.. _Apache-2.0: https://www.apache.org/licenses/LICENSE-2.0

.. </legal notes>



*)

METHOD lengthIsBetween
VAR_INPUT
	(* current string to check *)
	stringToCheck		:POINTER TO BYTE;
	(* lower limit of the string length *)
	minLength			:UDINT;
	(* upper limit of the string length *)
	maxLength			:UDINT;
	(* string length units of measurement *)
	stringLengthUnit	:UnicodeStringLengthUnit;
	(* message if the assertion is false *)
	message				:AssertMessage;
END_VAR
VAR
	(* length of current string to check in bytes *)
	stringToCheckByteCount		:UDINT;
	(* length of current string to check in characters *)
	stringToCheckCodePointCount	:UDINT;
	
	normalizedStringBuffer :POINTER TO BYTE; 
	bufferSize :UDINT;
	normalizedLength :UDINT;
	width :DINT;
	visibleCharacters :UDINT := 0;
END_VAR
VAR CONSTANT
	(*After decomposition one codepoint can extend up to 4 codepoints*)
	NORMALIZATION_FACTOR :UDINT := 4;
END_VAR
IF minLength > maxLength THEN
	THIS^.assertionWasWrong(message, THIS^.getDebugInfo('lengthIsBetween'));
	RETURN;
END_IF

CNM_UnicodeUtilities.GetUtf8StringLength(
	stringToCheck,
	byteCount => stringToCheckByteCount,
	characterCount => stringToCheckCodePointCount
);

// check if string is empty
IF (stringToCheckByteCount = 0) THEN
	IF (minLength > 0) THEN
		THIS^.assertionWasWrong(message, THIS^.getDebugInfo('lengthIsBetween'));
	END_IF
	RETURN;
END_IF

CASE (stringLengthUnit) OF
UnicodeStringLengthUnit.BYTES:
	IF (stringToCheckByteCount < minLength OR_ELSE stringToCheckByteCount > maxLength) THEN
		THIS^.assertionWasWrong(message, THIS^.getDebugInfo('lengthIsBetween'));
	END_IF

UnicodeStringLengthUnit.CHARACTERS:
	IF (stringToCheckCodePointCount < minLength OR_ELSE stringToCheckCodePointCount > maxLength) THEN
		THIS^.assertionWasWrong(message, THIS^.getDebugInfo('lengthIsBetween'));
	END_IF	
	
UnicodeStringLengthUnit.CHARACTERS_NFC:
	// string size cant increase with NFC
	normalizedStringBuffer := __NEW(BYTE, (stringToCheckByteCount + 1));
	IF normalizedStringBuffer = 0 THEN
		THIS^.assertionWasWrong(message, THIS^.getDebugInfo('lengthIsBetween, malloc failed'));
		RETURN;
	END_IF
	
	bufferSize := stringToCheckByteCount + 1; // stringsize + NULL terminator
	
	CNM_UnicodeUtilities.NormalizeUtf8String(
		utf8StringBuffer := stringToCheck,
		normalForm := CNM_UnicodeUtilities.NormalizationForm.NFC,
		normalizedStringBuffer := normalizedStringBuffer,
		bufferSize := bufferSize,
		normalizedStringLength => normalizedLength
	);
	
	CNM_UnicodeUtilities.GetUtf8StringLength(
		stringAddress := normalizedStringBuffer,
		characterCount => stringToCheckCodePointCount
	);
	
	__DELETE(normalizedStringBuffer);
	
	IF (stringToCheckCodePointCount < minLength OR_ELSE stringToCheckCodePointCount > maxLength) THEN
		THIS^.assertionWasWrong(message, THIS^.getDebugInfo('lengthIsBetween'));
	END_IF
	
UnicodeStringLengthUnit.CHARACTERS_NFD:
	// string size can increase with NFD
	normalizedStringBuffer := __NEW(BYTE, (stringToCheckByteCount * NORMALIZATION_FACTOR + 1));
	IF normalizedStringBuffer = 0 THEN
		THIS^.assertionWasWrong(message, THIS^.getDebugInfo('lengthIsBetween, malloc failed'));
		RETURN;
	END_IF
	
	bufferSize := stringToCheckByteCount * NORMALIZATION_FACTOR + 1; // stringsize (can increase for NFD) + NULL terminator
	
	CNM_UnicodeUtilities.NormalizeUtf8String(
		utf8StringBuffer := stringToCheck,
		normalForm := CNM_UnicodeUtilities.NormalizationForm.NFD,
		normalizedStringBuffer := normalizedStringBuffer,
		bufferSize := bufferSize,
		normalizedStringLength => normalizedLength
	);
	
	CNM_UnicodeUtilities.GetUtf8StringLength(
		stringAddress := normalizedStringBuffer,
		characterCount => stringToCheckCodePointCount
	);
	
	__DELETE(normalizedStringBuffer);
	
	IF (stringToCheckCodePointCount < minLength OR_ELSE stringToCheckCodePointCount > maxLength) THEN
		THIS^.assertionWasWrong(message, THIS^.getDebugInfo('lengthIsBetween'));
	END_IF
	
UnicodeStringLengthUnit.VISIBLE_CHARACTERS:
	CNM_UnicodeUtilities.GetUtf8StringWidth(stringToCheck, visibleCharacters => visibleCharacters);
	IF (visibleCharacters < minLength) OR_ELSE (visibleCharacters > maxLength) THEN
		THIS^.assertionWasWrong(message, THIS^.getDebugInfo('lengthIsBetween'));
	END_IF 
	
UnicodeStringLengthUnit.WIDTH:
	width := CNM_UnicodeUtilities.GetUtf8StringWidth(stringToCheck);
	IF ((
			width < 0
		) OR_ELSE (
			TO_UDINT(width) < minLength
		) OR_ELSE (
			TO_UDINT(width) > maxLength)
	) THEN
		THIS^.assertionWasWrong(message, THIS^.getDebugInfo('lengthIsBetween'));
	END_IF
ELSE
	; // do nothing
END_CASE
END_METHOD

(*

## Short summary
This assertion method checks if the current string ``stringToCheck`` length is equal to ``expectedLength``.
Processed strings must be in UTF-8 encoding

**Attention:** 
	All strings are handled as null-terminated byte streams

.. <legal notes>

legal notes
=================
| SPDX-FileCopyrightText: © 2024 ekvip automation GmbH <info@ekvip.de>
| SPDX-License-Identifier: Apache-2.0
| For details check: Apache-2.0_

.. _Apache-2.0: https://www.apache.org/licenses/LICENSE-2.0

.. </legal notes>



*)

METHOD lengthIsExact
VAR_INPUT
	(* current string to check *)
	stringToCheck		:POINTER TO BYTE;
	(* expected length of ``stringToCheck`` *)
	expectedLength		:UDINT;
	(* string length units of measurement *)
	stringLengthUnit	:UnicodeStringLengthUnit;
	(* message if the assertion is false *)
	message				:AssertMessage;
END_VAR
VAR
	(* length of current string to check in bytes *)
	stringToCheckByteCount		:UDINT;
	(* length of current string to check in characters *)
	stringToCheckCodePointCount	:UDINT;
	
	normalizedStringBuffer :POINTER TO BYTE; 
	bufferSize :UDINT;
	normalizedLength :UDINT;
	width :DINT;
	visibleCharacters :UDINT := 0;
END_VAR
VAR CONSTANT
	(*After decomposition one codepoint can extend up to 4 codepoints*)
	NORMALIZATION_FACTOR :UDINT := 4;
END_VAR
CNM_UnicodeUtilities.GetUtf8StringLength(
	stringToCheck,
	byteCount => stringToCheckByteCount,
	characterCount => stringToCheckCodePointCount
);

// check if string is empty
IF (stringToCheckByteCount = 0) THEN
	IF (expectedLength <> 0) THEN
		THIS^.assertionWasWrong(message, THIS^.getDebugInfo('LengthIsExact'));
	END_IF
	RETURN;
END_IF

CASE (stringLengthUnit) OF
UnicodeStringLengthUnit.BYTES:
	IF (stringToCheckByteCount <> expectedLength) THEN
		THIS^.assertionWasWrong(message, THIS^.getDebugInfo('LengthIsExact'));
	END_IF

UnicodeStringLengthUnit.CHARACTERS:
	IF (stringToCheckCodePointCount <> expectedLength) THEN
		THIS^.assertionWasWrong(message, THIS^.getDebugInfo('LengthIsExact'));
	END_IF	
	
UnicodeStringLengthUnit.CHARACTERS_NFC:
	// string size cant increase with NFC
	normalizedStringBuffer := __NEW(BYTE, (stringToCheckByteCount+1));
	IF normalizedStringBuffer = 0 THEN
		THIS^.assertionWasWrong(message, THIS^.getDebugInfo('lengthIsExact, malloc failed'));
		RETURN;
	END_IF
	bufferSize := stringToCheckByteCount + 1; // stringsize + NULL terminator
	
	CNM_UnicodeUtilities.NormalizeUtf8String(
		utf8StringBuffer := stringToCheck,
		normalForm := CNM_UnicodeUtilities.NormalizationForm.NFC,
		normalizedStringBuffer := normalizedStringBuffer,
		bufferSize := bufferSize,
		normalizedStringLength => normalizedLength
	);
	
	CNM_UnicodeUtilities.GetUtf8StringLength(
		stringAddress := normalizedStringBuffer,
		characterCount => stringToCheckCodePointCount
	);
	
	__DELETE(normalizedStringBuffer);
	
	IF (stringToCheckCodePointCount <> expectedLength) THEN
		THIS^.assertionWasWrong(message, THIS^.getDebugInfo('LengthIsExact'));
	END_IF
	
UnicodeStringLengthUnit.CHARACTERS_NFD:
	// string size can increase with NFD
	normalizedStringBuffer := __NEW(BYTE, (stringToCheckByteCount * NORMALIZATION_FACTOR + 1));
	IF normalizedStringBuffer = 0 THEN
		THIS^.assertionWasWrong(message, THIS^.getDebugInfo('lengthIsExact, malloc failed'));
		RETURN;
	END_IF
	bufferSize := stringToCheckByteCount * NORMALIZATION_FACTOR + 1; // stringsize can increase for NFD + NULL terminator
	
	CNM_UnicodeUtilities.NormalizeUtf8String(
		utf8StringBuffer := stringToCheck,
		normalForm := CNM_UnicodeUtilities.NormalizationForm.NFD,
		normalizedStringBuffer := normalizedStringBuffer,
		bufferSize := bufferSize,
		normalizedStringLength => normalizedLength
	);
	
	CNM_UnicodeUtilities.GetUtf8StringLength(
		stringAddress := normalizedStringBuffer,
		characterCount => stringToCheckCodePointCount
	);
	
	__DELETE(normalizedStringBuffer);
	
	IF (stringToCheckCodePointCount <> expectedLength) THEN
		THIS^.assertionWasWrong(message, THIS^.getDebugInfo('LengthIsExact'));
	END_IF
	
UnicodeStringLengthUnit.VISIBLE_CHARACTERS:
	CNM_UnicodeUtilities.GetUtf8StringWidth(stringToCheck, visibleCharacters => visibleCharacters);
	IF (visibleCharacters <> expectedLength) THEN
		THIS^.assertionWasWrong(message, THIS^.getDebugInfo('lengthIsExact'));
	END_IF
	
UnicodeStringLengthUnit.WIDTH:
	width := CNM_UnicodeUtilities.GetUtf8StringWidth(stringToCheck);
	IF ((width < 0) OR_ELSE (TO_UDINT(width) <> expectedLength)) THEN
		THIS^.assertionWasWrong(message, THIS^.getDebugInfo('LengthIsExact'));
	END_IF
ELSE
	; // do nothing
END_CASE
END_METHOD

(*

## Short summary
This assertion method checks if the current string ``stringToCheck`` length is equal or less than to ``maxLength``.
Processed strings must be in UTF-8 encoding

**Attention:** 
	All strings are handled as null-terminated byte streams

.. <legal notes>

legal notes
=================
| SPDX-FileCopyrightText: © 2024 ekvip automation GmbH <info@ekvip.de>
| SPDX-License-Identifier: Apache-2.0
| For details check: Apache-2.0_

.. _Apache-2.0: https://www.apache.org/licenses/LICENSE-2.0

.. </legal notes>



*)

METHOD lengthIsMax
VAR_INPUT
	(* current string to check *)
	stringToCheck		:POINTER TO BYTE;
	(* upper limit of the length of ``stringToCheck`` *)
	maxLength			:UDINT;
	(* string length units of measurement *)
	stringLengthUnit	:UnicodeStringLengthUnit;
	(* message if the assertion is false *)
	message				:AssertMessage;
END_VAR
VAR
	(* length of current string to check in bytes *)
	stringToCheckByteCount		:UDINT;
	(* length of current string to check in characters *)
	stringToCheckCodePointCount	:UDINT;
	
	normalizedStringBuffer :POINTER TO BYTE; 
	bufferSize :UDINT;
	normalizedLength :UDINT;
	width :DINT;
	visibleCharacters :UDINT := 0;
END_VAR
VAR CONSTANT
	(*After decomposition one codepoint can extend up to 4 codepoints*)
	NORMALIZATION_FACTOR :UDINT := 4;
END_VAR
CNM_UnicodeUtilities.GetUtf8StringLength(
	stringToCheck,
	byteCount => stringToCheckByteCount,
	characterCount => stringToCheckCodePointCount
);

// check if string is empty
RETURN (stringToCheckByteCount = 0);

CASE (stringLengthUnit) OF
UnicodeStringLengthUnit.BYTES:
	IF (stringToCheckByteCount > maxLength) THEN
		THIS^.assertionWasWrong(message, THIS^.getDebugInfo('LengthIsMax'));
	END_IF

UnicodeStringLengthUnit.CHARACTERS:
	IF (stringToCheckCodePointCount > maxLength) THEN
		THIS^.assertionWasWrong(message, THIS^.getDebugInfo('LengthIsMax'));
	END_IF	
	
UnicodeStringLengthUnit.CHARACTERS_NFC:
	// string size cant increase with NFC
	normalizedStringBuffer := __NEW(BYTE, (stringToCheckByteCount + 1));
	IF normalizedStringBuffer = 0 THEN
		THIS^.assertionWasWrong(message, THIS^.getDebugInfo('lengthIsMax, malloc failed'));
		RETURN;
	END_IF
	
	// stringsize + NULL terminator
	bufferSize := stringToCheckByteCount + 1; 
	
	CNM_UnicodeUtilities.NormalizeUtf8String(
		utf8StringBuffer := stringToCheck,
		normalForm := CNM_UnicodeUtilities.NormalizationForm.NFC,
		normalizedStringBuffer := normalizedStringBuffer,
		bufferSize := bufferSize,
		normalizedStringLength => normalizedLength
	);
	
	CNM_UnicodeUtilities.GetUtf8StringLength(
		stringAddress := normalizedStringBuffer,
		characterCount => stringToCheckCodePointCount
	);
	
	__DELETE(normalizedStringBuffer);
	
	IF (stringToCheckCodePointCount > maxLength) THEN
		THIS^.assertionWasWrong(message, THIS^.getDebugInfo('LengthIsMax'));
	END_IF
	
UnicodeStringLengthUnit.CHARACTERS_NFD:
	// string size can increase with NFD
	normalizedStringBuffer := __NEW(BYTE, (stringToCheckByteCount * NORMALIZATION_FACTOR + 1));
	IF normalizedStringBuffer = 0 THEN
		THIS^.assertionWasWrong(message, THIS^.getDebugInfo('lengthIsMax, malloc failed'));
		RETURN;
	END_IF
	bufferSize := stringToCheckByteCount * NORMALIZATION_FACTOR + 1; // stringsize can increase for NFD + NULL terminator
	
	CNM_UnicodeUtilities.NormalizeUtf8String(
		utf8StringBuffer := stringToCheck,
		normalForm := CNM_UnicodeUtilities.NormalizationForm.NFD,
		normalizedStringBuffer := normalizedStringBuffer,
		bufferSize := bufferSize,
		normalizedStringLength => normalizedLength
	);
	
	CNM_UnicodeUtilities.GetUtf8StringLength(
		stringAddress := normalizedStringBuffer,
		characterCount => stringToCheckCodePointCount
	);
	
	__DELETE(normalizedStringBuffer);
	
	IF (stringToCheckCodePointCount > maxLength) THEN
		THIS^.assertionWasWrong(message, THIS^.getDebugInfo('LengthIsMax'));
	END_IF
	
UnicodeStringLengthUnit.VISIBLE_CHARACTERS:
	CNM_UnicodeUtilities.GetUtf8StringWidth(stringToCheck, visibleCharacters => visibleCharacters);
	IF (visibleCharacters > maxLength) THEN
		THIS^.assertionWasWrong(message, THIS^.getDebugInfo('lengthIsMax'));
	END_IF
	
UnicodeStringLengthUnit.WIDTH:
	width := CNM_UnicodeUtilities.GetUtf8StringWidth(stringToCheck);
	IF ((width < 0) OR_ELSE (TO_UDINT(width) > maxLength)) THEN
		THIS^.assertionWasWrong(message, THIS^.getDebugInfo('LengthIsMax'));
	END_IF
ELSE
	; // do nothing
END_CASE
END_METHOD

(*

## Short summary
This assertion method checks if the current string ``stringToCheck`` length is equal or grater than to ``minLength``.
Processed strings must be in UTF-8 encoding

**Attention:** 
	All strings are handled as null-terminated byte streams

.. <legal notes>

legal notes
=================
| SPDX-FileCopyrightText: © 2024 ekvip automation GmbH <info@ekvip.de>
| SPDX-License-Identifier: Apache-2.0
| For details check: Apache-2.0_

.. _Apache-2.0: https://www.apache.org/licenses/LICENSE-2.0

.. </legal notes>



*)

METHOD lengthIsMin
VAR_INPUT
	(* current string to check *)
	stringToCheck		:POINTER TO BYTE;
	(* lower limit of the length of ``stringToCheck`` *)
	minLength			:UDINT;
	(* string length units of measurement *)
	stringLengthUnit	:UnicodeStringLengthUnit;
	(* message if the assertion is false *)
	message				:AssertMessage;
END_VAR
VAR
	(* length of current string to check in bytes *)
	stringToCheckByteCount		:UDINT;
	(* length of current string to check in characters *)
	stringToCheckCodePointCount	:UDINT;
	normalizedStringBuffer :POINTER TO BYTE; 
	bufferSize :UDINT;
	normalizedLength :UDINT;
	width :DINT;
	visibleCharacters :UDINT := 0;
END_VAR
VAR CONSTANT
	(*After decomposition one codepoint can extend up to 4 codepoints*)
	NORMALIZATION_FACTOR :UDINT := 4;
END_VAR
CNM_UnicodeUtilities.GetUtf8StringLength(
	stringToCheck,
	byteCount => stringToCheckByteCount,
	characterCount => stringToCheckCodePointCount
);

// check if string is empty
IF (stringToCheckByteCount = 0) THEN
	IF (minLength > 0) THEN
		THIS^.assertionWasWrong(message, THIS^.getDebugInfo('LengthIsMin'));
	END_IF
	RETURN;
END_IF

CASE (stringLengthUnit) OF
UnicodeStringLengthUnit.BYTES:
	IF (stringToCheckByteCount < minLength) THEN
		THIS^.assertionWasWrong(message, THIS^.getDebugInfo('LengthIsMin'));
	END_IF

UnicodeStringLengthUnit.CHARACTERS:
	IF (stringToCheckCodePointCount < minLength) THEN
		THIS^.assertionWasWrong(message, THIS^.getDebugInfo('LengthIsMin'));
	END_IF	
	
UnicodeStringLengthUnit.CHARACTERS_NFC:
	// string size cant increase with NFC
	normalizedStringBuffer := __NEW(BYTE, (stringToCheckByteCount + 1));
	IF normalizedStringBuffer = 0 THEN
		THIS^.assertionWasWrong(message, THIS^.getDebugInfo('lengthIsMin, malloc failed'));
		RETURN;
	END_IF
	bufferSize := stringToCheckByteCount + 1; // stringsize + NULL terminator
	
	CNM_UnicodeUtilities.NormalizeUtf8String(
		utf8StringBuffer := stringToCheck,
		normalForm := CNM_UnicodeUtilities.NormalizationForm.NFC,
		normalizedStringBuffer := normalizedStringBuffer,
		bufferSize := bufferSize,
		normalizedStringLength => normalizedLength
	);
	
	CNM_UnicodeUtilities.GetUtf8StringLength(
		stringAddress := normalizedStringBuffer,
		characterCount => stringToCheckCodePointCount
	);
	
	__DELETE(normalizedStringBuffer);
	
	IF (stringToCheckCodePointCount < minLength) THEN
		THIS^.assertionWasWrong(message, THIS^.getDebugInfo('LengthIsMin'));
	END_IF
	
UnicodeStringLengthUnit.CHARACTERS_NFD:
	// string size can increase with NFD
	normalizedStringBuffer := __NEW(BYTE, (stringToCheckByteCount * NORMALIZATION_FACTOR + 1));
	IF normalizedStringBuffer = 0 THEN
		THIS^.assertionWasWrong(message, THIS^.getDebugInfo('lengthIsMin, malloc failed'));
		RETURN;
	END_IF
	bufferSize := stringToCheckByteCount * NORMALIZATION_FACTOR + 1; // stringsize can increase for NFD + NULL terminator
	
	CNM_UnicodeUtilities.NormalizeUtf8String(
		utf8StringBuffer := stringToCheck,
		normalForm := CNM_UnicodeUtilities.NormalizationForm.NFD,
		normalizedStringBuffer := normalizedStringBuffer,
		bufferSize := bufferSize,
		normalizedStringLength => normalizedLength
	);
	
	CNM_UnicodeUtilities.GetUtf8StringLength(
		stringAddress := normalizedStringBuffer,
		characterCount => stringToCheckCodePointCount
	);
	
	__DELETE(normalizedStringBuffer);
	
	IF (stringToCheckCodePointCount < minLength) THEN
		THIS^.assertionWasWrong(message, THIS^.getDebugInfo('LengthIsMin'));
	END_IF
	
UnicodeStringLengthUnit.VISIBLE_CHARACTERS:
	CNM_UnicodeUtilities.GetUtf8StringWidth(stringToCheck, visibleCharacters => visibleCharacters);
	IF (visibleCharacters < minLength)THEN
		THIS^.assertionWasWrong(message, THIS^.getDebugInfo('lengthIsMin'));
	END_IF
	
UnicodeStringLengthUnit.WIDTH:
	width := CNM_UnicodeUtilities.GetUtf8StringWidth(stringToCheck);
	IF ((width < 0) OR_ELSE (TO_UDINT(width) < minLength)) THEN
		THIS^.assertionWasWrong(message, THIS^.getDebugInfo('LengthIsMin'));
	END_IF
ELSE
	; // do nothing
END_CASE
END_METHOD

(*

## Short summary
This assertion method checks if the current string ``stringToCheck`` starts with string ``start``.
Processed strings must be in UTF-8 encoding

**Attention:** 
	All strings are handled as null-terminated byte streams

.. <legal notes>

legal notes
=================
| SPDX-FileCopyrightText: © 2024 ekvip automation GmbH <info@ekvip.de>
| SPDX-License-Identifier: Apache-2.0
| For details check: Apache-2.0_

.. _Apache-2.0: https://www.apache.org/licenses/LICENSE-2.0

.. </legal notes>



*)

METHOD startsWith
VAR_INPUT
	(* current string to check *)
	stringToCheck	:POINTER TO BYTE;
	(* expected start of ``stringToCheck`` *)
	start			:POINTER TO BYTE;
	(* ``TRUE`` means ignore cases; ``FALSE`` means that cases must be equal too *)
	ignoreCases		:BOOL;
	(* ``TRUE`` means truncation of spaces on the left side of ``stringToCheck``*)
	trim		:BOOL;
	(* message if the assertion is false *)
	message			:AssertMessage;
	(*normalize both strings for check*)
	normalizeStrings :BOOL := TRUE;
END_VAR
VAR
	(* length of ``stringToCheck`` in bytes *)
	lengthStringToCheckInByte	:UDINT;	
	(* length of ``searchString`` in bytes *)
	lengthSearchStringInByte	:UDINT;
	(* DWORD array we use to check *)
	usedCodePointsToCheck, normalizedUsedCodePointsToCheck :POINTER TO CNM_UnicodeUtilities.UnicodeCodePoint;
	usedCodePointToCheckCount	:UDINT;
	
	(* DWORD array we use to compare *)
	usedStartCodePoints, normalizedUsedStartCodePoints :POINTER TO CNM_UnicodeUtilities.UnicodeCodePoint;
	usedStartCodePointCount		:UDINT;
END_VAR
VAR CONSTANT
	(*After decomposition one codepoint can extend up to 4 codepoints*)
	NORMALIZATION_FACTOR :UDINT := 4;
END_VAR
CNM_UnicodeUtilities.GetUtf8StringLength(stringAddress := stringToCheck, byteCount => lengthStringToCheckInByte);
CNM_UnicodeUtilities.GetUtf8StringLength(stringAddress := start, byteCount => lengthSearchStringInByte);

IF (((
		NOT normalizeStrings 
	) OR ( 
		lengthStringToCheckInByte = 0
	) OR (
		lengthSearchStringInByte = 0
	)) AND_THEN(
		NOT THIS^.isContainsCheckNecessary(
			stringToCheck		:= stringToCheck,
			searchString		:= start,
			lengthStringToCheck	:= lengthStringToCheckInByte,
			lengthSearchString	:= lengthSearchStringInByte,
			additionalText		:= THIS^.getDebugInfo('startsWith'),
			message				:= message
		) 
	)
) THEN
	RETURN;
END_IF

usedCodePointsToCheck := __NEW(CNM_UnicodeUtilities.UnicodeCodePoint, lengthStringToCheckInByte);
IF (usedCodePointsToCheck = 0) THEN
	THIS^.assertionWasWrong(message, THIS^.getDebugInfo('startsWith, malloc failed'));
	RETURN;
END_IF

usedStartCodePoints := __NEW(CNM_UnicodeUtilities.UnicodeCodePoint, lengthSearchStringInByte);
IF (usedStartCodePoints = 0) THEN
	__DELETE(usedCodePointsToCheck);
	THIS^.assertionWasWrong(message, THIS^.getDebugInfo('startsWith, malloc failed'));
	RETURN;
END_IF

(* convert ``stringToCheck`` to code points *)
CNM_UnicodeUtilities.GetCodepointsFromUtf8String(
	utf8StringAddress := stringToCheck, 
	utf8StringByteCount := lengthStringToCheckInByte, 
	codePointBuffer := usedCodePointsToCheck,
	bufferSize := SIZEOF(CNM_UnicodeUtilities.UnicodeCodePoint)*lengthStringToCheckInByte, 
	codePointsCount => usedCodePointToCheckCount);

(* convert ``searchString`` to code points *)
CNM_UnicodeUtilities.GetCodepointsFromUtf8String(
	utf8StringAddress 	:= start, 
	utf8StringByteCount := lengthSearchStringInByte, 
	codePointBuffer	:= usedStartCodePoints,
	bufferSize := SIZEOF(CNM_UnicodeUtilities.UnicodeCodePoint)*lengthSearchStringInByte,
	codePointsCount => usedStartCodePointCount);



IF normalizeStrings THEN
	normalizedUsedCodePointsToCheck := __NEW(
		CNM_UnicodeUtilities.UnicodeCodePoint,
		(lengthStringToCheckInByte * NORMALIZATION_FACTOR)
	);
	IF (normalizedUsedCodePointsToCheck = 0) THEN
		THIS^.assertionWasWrong(message, THIS^.getDebugInfo('startsWith, malloc failed'));
		__DELETE(usedCodePointsToCheck);
		__DELETE(usedStartCodePoints);
		RETURN;
	END_IF
	normalizedUsedStartCodePoints := __NEW(
		CNM_UnicodeUtilities.UnicodeCodePoint,
		(lengthSearchStringInByte * NORMALIZATION_FACTOR)
	);
	IF (normalizedUsedStartCodePoints = 0) THEN
		THIS^.assertionWasWrong(message, THIS^.getDebugInfo('startsWith, malloc failed'));
		__DELETE(usedCodePointsToCheck);
		__DELETE(usedStartCodePoints);
		__DELETE(normalizedUsedCodePointsToCheck);	
		RETURN;
	END_IF

	CNM_UnicodeUtilities.NormalizeCodepointsFormD(
		codePoints := usedCodePointsToCheck,
		codePointsCount := usedCodePointToCheckCount,
		normalizedCodepoints := normalizedUsedCodePointsToCheck,
		bufferSize := (lengthStringToCheckInByte * NORMALIZATION_FACTOR) * SIZEOF(CNM_UnicodeUtilities.UnicodeCodePoint),
		normalizedCodepointsCount => usedCodePointToCheckCount
	);
	__DELETE(usedCodePointsToCheck);
	usedCodePointsToCheck := normalizedUsedCodePointsToCheck;
	
	CNM_UnicodeUtilities.NormalizeCodepointsFormD(
		codePoints := usedStartCodePoints,
		codePointsCount := usedStartCodePointCount,
		normalizedCodepoints := normalizedUsedStartCodePoints,
		bufferSize := (lengthSearchStringInByte * NORMALIZATION_FACTOR) * SIZEOF(CNM_UnicodeUtilities.UnicodeCodePoint),
		normalizedCodepointsCount => usedStartCodePointCount
	);
	__DELETE(usedStartCodePoints);
	usedStartCodePoints := normalizedUsedStartCodePoints;
END_IF

IF (trim) THEN
	CNM_UnicodeUtilities.TrimLeftCodepoints(
		codepoints := usedStartCodePoints,
		codepointCount := usedStartCodePointCount,
		newCodepointCount => usedStartCodePointCount
	);
	CNM_UnicodeUtilities.TrimLeftCodepoints(
		codepoints := usedCodePointsToCheck,
		codepointCount := usedCodePointToCheckCount,
		newCodepointCount => usedCodePointToCheckCount
	);
END_IF

IF (ignoreCases) THEN
	CNM_UnicodeUtilities.GetUpperCaseForCodepoint(usedCodePointsToCheck, usedCodePointToCheckCount);
	CNM_UnicodeUtilities.GetUpperCaseForCodepoint(usedStartCodePoints, usedStartCodePointCount);
END_IF

IF (Tc2_System.MEMCMP(
		usedCodePointsToCheck,
		usedStartCodePoints, 
		usedStartCodePointCount*SIZEOF(CNM_UnicodeUtilities.UnicodeCodePoint)
	) <> CNM_ReturnTypes.ComparationResult.EQUAL
) THEN
	THIS^.assertionWasWrong(message, THIS^.getDebugInfo('startsWith'));
END_IF;

__DELETE(usedCodePointsToCheck);
__DELETE(usedStartCodePoints);
END_METHOD

END_FUNCTION_BLOCK

// ---- Assertor/Assertions/StringAssertion/Unicode/Classes/UnicodeAssertions.TcPOU
(*

## Short summary
Class provides assert statements
for UTF-8 and UTF-16 strings with an undefined length.

**Attention:** 
	All strings are handled as null terminated byte/word streams.
	For UTF-8 is end of the string 16#00
	For UTF-16 is end of the string 16#00_00

**Attention:** 
	The interface `IUnicodeAssertions` uses ``ANY_STRING``, 
	for this it's not possible to use literals/constants,
	because for ``ANY`` types generates the compiler ``__SYSTEM.AnyType``
	and ``__SYSTEM.AnyType`` contains a pointer  

.. <legal notes>

legal notes
=================
| SPDX-FileCopyrightText: © 2022 ekvip automation GmbH <info@ekvip.de>
| SPDX-License-Identifier: Apache-2.0
| For details check: Apache-2.0_

.. _Apache-2.0: https://www.apache.org/licenses/LICENSE-2.0

.. </legal notes>



*)

{attribute 'reflection'}
FUNCTION_BLOCK INTERNAL UnicodeAssertions EXTENDS AbstractAssertion IMPLEMENTS IUnicodeStringAssertions
VAR
	(* class to handle the utf 8 string assertions *)  
	utf8Assertions	:Utf8StringPointerAssertions();
	(* class to handle the utf 16 string assertions *)  
	utf16Assertions		:Utf16StringPointerAssertions();	
END_VAR

(*

## Short summary
This abstract property returns the class name of the concrete object, 
It's for debugging purpose

.. <legal notes>

legal notes
=================
| SPDX-FileCopyrightText: © 2022 ekvip automation GmbH <info@ekvip.de>
| SPDX-License-Identifier: Apache-2.0
| For details check: Apache-2.0_

.. _Apache-2.0: https://www.apache.org/licenses/LICENSE-2.0

.. </legal notes>

*)

PROPERTY className :CNM_AbstractObject.ClassName
GET
className := 'CNM_Assertor.UnicodeAssertions';
END_GET
END_PROPERTY

(*

## Short summary
This assertion method checks if the current string ``stringToCheck`` contains the search string

**Attention:** 
	All strings are handled as null terminated byte/word streams.
	For UTF-8 is end of the string 16#00
	For UTF-16 is end of the string 16#00_00

**Attention:** 
	The interface `IUnicodeAssertions` uses ``ANY_STRING``, 
	for this it's not possible to use literals/constants,
	because for ``ANY`` types generates the compiler ``__SYSTEM.AnyType``
	and ``__SYSTEM.AnyType`` contains a pointer  

.. <legal notes>

legal notes
=================
| SPDX-FileCopyrightText: © 2022 ekvip automation GmbH <info@ekvip.de>
| SPDX-License-Identifier: Apache-2.0
| For details check: Apache-2.0_

.. _Apache-2.0: https://www.apache.org/licenses/LICENSE-2.0

.. </legal notes>



*)

METHOD contains
VAR_INPUT
	(* current string to check *)
	stringToCheck	:ANY_STRING;
	(* string must be found in ``stringToCheck`` *)
	searchString	:ANY_STRING;
	(* message if the assertion is false *)
	message			:AssertMessage;
	(* ``TRUE`` means ignore cases; ``FALSE`` means cases must be equal too *)
	ignoreCases		:BOOL := FALSE;
	(*normalize both strings for check*)
	normalizeStrings :BOOL := TRUE;
END_VAR
IF ((
		stringToCheck.TypeClass <> searchString.TypeClass
	) OR_ELSE (
		stringToCheck.diSize = 0 
	) OR_ELSE ( 
		searchString.diSize = 0 
	)
) THEN
	THIS^.assertionWasWrong(message, THIS^.getDebugInfo('contains'));
	RETURN;
END_IF

CASE stringToCheck.TypeClass OF
TYPE_CLASS.TYPE_STRING:
	THIS^.utf8Assertions.contains(
		stringToCheck := stringToCheck.pValue,
		searchString := searchString.pValue,
		ignoreCases := ignoreCases,
		message := message
	);
TYPE_CLASS.TYPE_WSTRING:
	THIS^.utf16Assertions.contains(
		stringToCheck := stringToCheck.pValue,
		searchString := searchString.pValue,
		ignoreCases := ignoreCases,
		message := message,
		normalizeStrings := normalizeStrings
	);
ELSE
	; // do nothing
END_CASE
END_METHOD

(*

## Short summary
This assertion method checks if the current string ``stringToCheck`` not contains the search string

**Attention:** 
	All strings are handled as null terminated byte/word streams.
	For UTF-8 is end of the string 16#00
	For UTF-16 is end of the string 16#00_00

**Attention:** 
	The interface `IUnicodeAssertions` uses ``ANY_STRING``, 
	for this it's not possible to use literals/constants,
	because for ``ANY`` types generates the compiler ``__SYSTEM.AnyType``
	and ``__SYSTEM.AnyType`` contains a pointer  

.. <legal notes>

legal notes
=================
| SPDX-FileCopyrightText: © 2022 ekvip automation GmbH <info@ekvip.de>
| SPDX-License-Identifier: Apache-2.0
| For details check: Apache-2.0_

.. _Apache-2.0: https://www.apache.org/licenses/LICENSE-2.0

.. </legal notes>



*)

METHOD containsNo
VAR_INPUT
	(* current string to check *)
	stringToCheck	:ANY_STRING;
	(* string that must not be found in ``stringToCheck`` *)
	searchString	:ANY_STRING;
	(* message if the assertion is false *)
	message			:AssertMessage;
	(* ``TRUE`` means ignore cases; ``FALSE`` means cases must be equal too *)
	ignoreCases		:BOOL := FALSE;
	(*normalize both strings for check*)
	normalizeStrings :BOOL := TRUE;
END_VAR
IF ((
		stringToCheck.TypeClass <> searchString.TypeClass
	) OR_ELSE ( 
		stringToCheck.diSize = 0 
	) OR_ELSE ( 
		searchString.diSize = 0 
	)
) THEN
	THIS^.assertionWasWrong(message, THIS^.getDebugInfo('containsNo'));
	RETURN;
END_IF

CASE stringToCheck.TypeClass OF
TYPE_CLASS.TYPE_STRING:
	THIS^.utf8Assertions.containsNo(
		stringToCheck := stringToCheck.pValue,
		searchString := searchString.pValue,
		ignoreCases := ignoreCases,
		message := message
	);
TYPE_CLASS.TYPE_WSTRING:
	THIS^.utf16Assertions.containsNo(
		stringToCheck := stringToCheck.pValue,
		searchString := searchString.pValue,
		ignoreCases := ignoreCases,
		message := message,
		normalizeStrings := normalizeStrings
	);
ELSE
	; // do nothing
END_CASE
END_METHOD

(*

## Short summary
This assertion method checks if the current string ``stringToCheck`` ends with ``end``

**Attention:** 
	All strings are handled as null terminated byte/word streams.
	For UTF-8 is end of the string 16#00
	For UTF-16 is end of the string 16#00_00

**Attention:** 
	The interface `IUnicodeAssertions` uses ``ANY_STRING``, 
	for this it's not possible to use literals/constants,
	because for ``ANY`` types generates the compiler ``__SYSTEM.AnyType``
	and ``__SYSTEM.AnyType`` contains a pointer  

**Attention:** 
	end of the string is **ALWAYS** the right side of the string 
	even for writings which written from right to left like Hebrew or Arabic

.. <legal notes>

legal notes
=================
| SPDX-FileCopyrightText: © 2022 ekvip automation GmbH <info@ekvip.de>
| SPDX-License-Identifier: Apache-2.0
| For details check: Apache-2.0_

.. _Apache-2.0: https://www.apache.org/licenses/LICENSE-2.0

.. </legal notes>



*)

METHOD endsWith
VAR_INPUT
	(* current string to check *)
	stringToCheck	:ANY_STRING;
	(* expected end of ``stringToCheck`` *)
	end				:ANY_STRING;
	(* message if the assertion is false *)
	message			:AssertMessage;
	(* ``TRUE`` means ignore cases; ``FALSE`` means cases must be equal too *)
	ignoreCases		:BOOL := FALSE;
	(* ``TRUE`` means truncation of spaces on the right side of ``stringToCheck``*)
	trim			:BOOL := FALSE;
	(*normalize both strings for check*)
	normalizeStrings :BOOL := TRUE;
END_VAR
IF ((
		stringToCheck.TypeClass <> end.TypeClass
	) OR_ELSE (
		 stringToCheck.diSize = 0
	) OR_ELSE (
		 end.diSize = 0
	)
) THEN
	THIS^.assertionWasWrong(message, THIS^.getDebugInfo('endsWith'));
	RETURN;
END_IF

CASE stringToCheck.TypeClass OF
TYPE_CLASS.TYPE_STRING:
	THIS^.utf8Assertions.endsWith(
		stringToCheck := stringToCheck.pValue,
		end := end.pValue,
		ignoreCases := ignoreCases,
		trim := trim,
		message := message,
		normalizeStrings := normalizeStrings
	);
TYPE_CLASS.TYPE_WSTRING:
	THIS^.utf16Assertions.endsWith(
		stringToCheck := stringToCheck.pValue,
		end := end.pValue,
		ignoreCases := ignoreCases,
		trim := trim,
		message := message,
		normalizeStrings := normalizeStrings
	);
ELSE
	; // do nothing
END_CASE
END_METHOD

(*

## Short summary
This assertion method checks if the current string ``stringToCheck`` is empty

**Attention:** 
	All strings are handled as null terminated byte/word streams.
	For UTF-8 is end of the string 16#00
	For UTF-16 is end of the string 16#00_00

**Attention:** 
	The interface `IUnicodeAssertions` uses ``ANY_STRING``, 
	for this it's not possible to use literals/constants,
	because for ``ANY`` types generates the compiler ``__SYSTEM.AnyType``
	and ``__SYSTEM.AnyType`` contains a pointer  

.. <legal notes>

legal notes
=================
| SPDX-FileCopyrightText: © 2022 ekvip automation GmbH <info@ekvip.de>
| SPDX-License-Identifier: Apache-2.0
| For details check: Apache-2.0_

.. _Apache-2.0: https://www.apache.org/licenses/LICENSE-2.0

.. </legal notes>



*)

METHOD isEmpty
VAR_INPUT
	(* current string to check *)
	stringToCheck	:ANY_STRING;
	(* message if the assertion is false *)
	message			:AssertMessage;
END_VAR
VAR CONSTANT
	(* strings are null terminated *)
	END_OF_UTF8_STRING	:BYTE := 16#00;
	(* strings are null terminated *)
	END_OF_UTF16_STRING	:WORD := 16#0000;
END_VAR
CASE stringToCheck.TypeClass OF
TYPE_CLASS.TYPE_STRING:
	IF (stringToCheck.pValue^ <> END_OF_UTF8_STRING) THEN
		THIS^.assertionWasWrong(message, THIS^.getDebugInfo('isEmpty'));
	END_IF
TYPE_CLASS.TYPE_WSTRING:
	IF (stringToCheck.pValue^ <> END_OF_UTF16_STRING) THEN
		THIS^.assertionWasWrong(message, THIS^.getDebugInfo('isEmpty'));
	END_IF
ELSE
	; // do nothing
END_CASE
END_METHOD

(*

## Short summary
This assertion method checks if the current string ``stringToCheck`` is equal to ``expected``

**Attention:** 
	All strings are handled as null terminated byte/word streams.
	For UTF-8 is end of the string 16#00
	For UTF-16 is end of the string 16#00_00

**Attention:** 
	The interface `IUnicodeAssertions` uses ``ANY_STRING``, 
	for this it's not possible to use literals/constants,
	because for ``ANY`` types generates the compiler ``__SYSTEM.AnyType``
	and ``__SYSTEM.AnyType`` contains a pointer  

.. <legal notes>

legal notes
=================
| SPDX-FileCopyrightText: © 2022 ekvip automation GmbH <info@ekvip.de>
| SPDX-License-Identifier: Apache-2.0
| For details check: Apache-2.0_

.. _Apache-2.0: https://www.apache.org/licenses/LICENSE-2.0

.. </legal notes>



*)

METHOD isEqualTo
VAR_INPUT
	(* current string to check *)
	stringToCheck	:ANY_STRING;
	(* ``stringToCheck`` must be equal to expected *)
	expected		:ANY_STRING;
	(* message if the assertion is false *)
	message			:AssertMessage;
	(* ``TRUE`` means ignore cases; ``FALSE`` means cases must be equal too *)
	ignoreCases		:BOOL := FALSE;
	(*normalize both strings for check*)
	normalizeStrings :BOOL := TRUE;
END_VAR
IF ((
		stringToCheck.TypeClass <> expected.TypeClass
	) OR_ELSE ( 
		stringToCheck.diSize = 0
	) OR_ELSE ( 
		expected.diSize = 0 
	)
) THEN
	THIS^.assertionWasWrong(message, THIS^.getDebugInfo('isEqualTo'));
	RETURN;
END_IF

CASE stringToCheck.TypeClass OF
TYPE_CLASS.TYPE_STRING:
	THIS^.utf8Assertions.isEqualTo(
		stringToCheck := stringToCheck.pValue,
		expected := expected.pValue,
		ignoreCases := ignoreCases,
		message := message
	);
TYPE_CLASS.TYPE_WSTRING:
	THIS^.utf16Assertions.isEqualTo(
		stringToCheck := stringToCheck.pValue,
		expected := expected.pValue,
		ignoreCases := ignoreCases,
		message := message,
		normalizeStrings := normalizeStrings
	);	
ELSE
	; // do nothing
END_CASE
END_METHOD

(*

## Short summary
This assertion method checks if the current string ``stringToCheck`` is not empty

**Attention:** 
	All strings are handled as null terminated byte/word streams.
	For UTF-8 is end of the string 16#00
	For UTF-16 is end of the string 16#00_00

**Attention:** 
	The interface `IUnicodeAssertions` uses ``ANY_STRING``, 
	for this it's not possible to use literals/constants,
	because for ``ANY`` types generates the compiler ``__SYSTEM.AnyType``
	and ``__SYSTEM.AnyType`` contains a pointer  

.. <legal notes>

legal notes
=================
| SPDX-FileCopyrightText: © 2022 ekvip automation GmbH <info@ekvip.de>
| SPDX-License-Identifier: Apache-2.0
| For details check: Apache-2.0_

.. _Apache-2.0: https://www.apache.org/licenses/LICENSE-2.0

.. </legal notes>



*)

METHOD isNotEmpty
VAR_INPUT
	(* current string to check *)
	stringToCheck	:ANY_STRING;
	(* message if the assertion is false *)
	message			:AssertMessage;
END_VAR
VAR CONSTANT
	(* strings are null terminated *)
	END_OF_UTF8_STRING	:BYTE := 16#00;
	(* strings are null terminated *)
	END_OF_UTF16_STRING	:WORD := 16#0000;
END_VAR
CASE stringToCheck.TypeClass OF
TYPE_CLASS.TYPE_STRING:
	IF (stringToCheck.pValue^ = END_OF_UTF8_STRING) THEN
		THIS^.assertionWasWrong(message, THIS^.getDebugInfo('isNotEmpty'));
	END_IF
TYPE_CLASS.TYPE_WSTRING:
	IF (stringToCheck.pValue^ = END_OF_UTF16_STRING) THEN
		THIS^.assertionWasWrong(message, THIS^.getDebugInfo('isNotEmpty'));
	END_IF
ELSE
	; // do nothing
END_CASE
END_METHOD

(*

## Short summary
This assertion method checks if the current string ``stringToCheck`` is not equal to ``unexpected``

**Attention:** 
	All strings are handled as null terminated byte/word streams.
	For UTF-8 is end of the string 16#00
	For UTF-16 is end of the string 16#00_00

**Attention:** 
	The interface `IUnicodeAssertions` uses ``ANY_STRING``, 
	for this it's not possible to use literals/constants,
	because for ``ANY`` types generates the compiler ``__SYSTEM.AnyType``
	and ``__SYSTEM.AnyType`` contains a pointer  

.. <legal notes>

legal notes
=================
| SPDX-FileCopyrightText: © 2022 ekvip automation GmbH <info@ekvip.de>
| SPDX-License-Identifier: Apache-2.0
| For details check: Apache-2.0_

.. _Apache-2.0: https://www.apache.org/licenses/LICENSE-2.0

.. </legal notes>



*)

METHOD isNotEqualTo
VAR_INPUT
	(* current string to check *)
	stringToCheck	:ANY_STRING;
	(* ``stringToCheck`` must be not equal to expected *)
	unexpected		:ANY_STRING;
	(* message if the assertion is false *)
	message			:AssertMessage;
	(* ``TRUE`` means ignore cases; ``FALSE`` means cases must be equal too *)
	ignoreCases		:BOOL := FALSE;
	(*normalize both strings for check*)
	normalizeStrings :BOOL := TRUE;
END_VAR
IF ((
		stringToCheck.TypeClass <> unexpected.TypeClass
	) OR_ELSE ( 
		stringToCheck.diSize = 0 
	) OR_ELSE ( 
		unexpected.diSize = 0 
	)
) THEN
	THIS^.assertionWasWrong(message, THIS^.getDebugInfo('isNotEqualTo'));
	RETURN;
END_IF

CASE stringToCheck.TypeClass OF
TYPE_CLASS.TYPE_STRING:
	THIS^.utf8Assertions.isNotEqualTo(
		stringToCheck := stringToCheck.pValue,
		unexpected := unexpected.pValue,
		ignoreCases := ignoreCases,
		message := message
	);
TYPE_CLASS.TYPE_WSTRING:
	THIS^.utf16Assertions.isNotEqualTo(
		stringToCheck := stringToCheck.pValue,
		unexpected := unexpected.pValue,
		ignoreCases := ignoreCases,
		message := message,
		normalizeStrings := normalizeStrings
	);	
ELSE
	; // do nothing
END_CASE
END_METHOD

(*

## Short summary
This assertion method checks if the current string ``stringToCheck`` is length
is between ``minLength`` and ``maxLength``

**Attention:** 
	All strings are handled as null terminated byte/word streams.
	For UTF-8 is end of the string 16#00
	For UTF-16 is end of the string 16#00_00

**Attention:** 
	The interface `IUnicodeAssertions` uses ``ANY_STRING``, 
	for this it's not possible to use literals/constants,
	because for ``ANY`` types generates the compiler ``__SYSTEM.AnyType``
	and ``__SYSTEM.AnyType`` contains a pointer  

.. <legal notes>

legal notes
=================
| SPDX-FileCopyrightText: © 2022 ekvip automation GmbH <info@ekvip.de>
| SPDX-License-Identifier: Apache-2.0
| For details check: Apache-2.0_

.. _Apache-2.0: https://www.apache.org/licenses/LICENSE-2.0

.. </legal notes>



*)

METHOD lengthIsBetween
VAR_INPUT
	(* current string to check *)
	stringToCheck	:ANY_STRING;
	(* lower limit of the string length *)
	minLength		:UDINT;
	(* upper limit of the string length *)
	maxLength		:UDINT;
	(* string length units of measurement *)
	stringLengthUnit	:UnicodeStringLengthUnit;
	(* message if the assertion is false *)
	message			:AssertMessage;
END_VAR
CASE stringToCheck.TypeClass OF
TYPE_CLASS.TYPE_STRING:
	THIS^.utf8Assertions.lengthIsBetween(
		stringToCheck	:= stringToCheck.pValue,
		minLength		:= minLength,
		maxLength		:= maxLength,
		stringLengthUnit := stringLengthUnit,
		message			:= message		
	);
TYPE_CLASS.TYPE_WSTRING:
	THIS^.utf16Assertions.lengthIsBetween(
		stringToCheck	:= stringToCheck.pValue,
		minLength		:= minLength,
		maxLength		:= maxLength,
		stringLengthUnit := stringLengthUnit,
		message			:= message
	);
ELSE
	; // do nothing
END_CASE
END_METHOD

(*

## Short summary
This assertion method checks if the current string ``stringToCheck`` is length
is equal to ``expectedLength``

**Attention:** 
	All strings are handled as null terminated byte/word streams.
	For UTF-8 is end of the string 16#00
	For UTF-16 is end of the string 16#00_00

**Attention:** 
	The interface `IUnicodeAssertions` uses ``ANY_STRING``, 
	for this it's not possible to use literals/constants,
	because for ``ANY`` types generates the compiler ``__SYSTEM.AnyType``
	and ``__SYSTEM.AnyType`` contains a pointer  

.. <legal notes>

legal notes
=================
| SPDX-FileCopyrightText: © 2022 ekvip automation GmbH <info@ekvip.de>
| SPDX-License-Identifier: Apache-2.0
| For details check: Apache-2.0_

.. _Apache-2.0: https://www.apache.org/licenses/LICENSE-2.0

.. </legal notes>



*)

METHOD lengthIsExact
VAR_INPUT
	(* current string to check *)
	stringToCheck	:ANY_STRING;
	(* expected length of ``stringToCheck`` *)
	expectedLength	:UDINT;
	(* string length units of measurement *)
	stringLengthUnit	:UnicodeStringLengthUnit;
	(* message if the assertion is false *)
	message			:AssertMessage;
END_VAR
CASE stringToCheck.TypeClass OF
TYPE_CLASS.TYPE_STRING:
	THIS^.utf8Assertions.lengthIsExact(
		stringToCheck	:= stringToCheck.pValue,
		expectedLength	:= expectedLength,
		stringLengthUnit := stringLengthUnit,
		message			:= message
	);
TYPE_CLASS.TYPE_WSTRING:
	THIS^.utf16Assertions.lengthIsExact(
		stringToCheck	:= stringToCheck.pValue,
		expectedLength	:= expectedLength,
		stringLengthUnit := stringLengthUnit,
		message			:= message
	);
ELSE
	; // do nothing
END_CASE
END_METHOD

(*

## Short summary
This assertion method checks if the current string ``stringToCheck`` is length
is equal or less than to ``maxLength``

**Attention:** 
	All strings are handled as null terminated byte/word streams.
	For UTF-8 is end of the string 16#00
	For UTF-16 is end of the string 16#00_00

**Attention:** 
	The interface `IUnicodeAssertions` uses ``ANY_STRING``, 
	for this it's not possible to use literals/constants,
	because for ``ANY`` types generates the compiler ``__SYSTEM.AnyType``
	and ``__SYSTEM.AnyType`` contains a pointer   

.. <legal notes>

legal notes
=================
| SPDX-FileCopyrightText: © 2022 ekvip automation GmbH <info@ekvip.de>
| SPDX-License-Identifier: Apache-2.0
| For details check: Apache-2.0_

.. _Apache-2.0: https://www.apache.org/licenses/LICENSE-2.0

.. </legal notes>



*)

METHOD lengthIsMax
VAR_INPUT
	(* current string to check *)
	stringToCheck	:ANY_STRING;
	(* upper limit of the length of ``stringToCheck`` *)
	maxLength		:UDINT;
	(* string length units of measurement *)
	stringLengthUnit	:UnicodeStringLengthUnit;
	(* message if the assertion is false *)
	message			:AssertMessage;
END_VAR
CASE stringToCheck.TypeClass OF
TYPE_CLASS.TYPE_STRING:
	THIS^.utf8Assertions.lengthIsMax(
		stringToCheck	:= stringToCheck.pValue,
		maxLength		:= maxLength,
		stringLengthUnit := stringLengthUnit,
		message			:= message
	);
TYPE_CLASS.TYPE_WSTRING:
	THIS^.utf16Assertions.lengthIsMax(
		stringToCheck	:= stringToCheck.pValue,
		maxLength		:= maxLength,
		stringLengthUnit := stringLengthUnit,
		message			:= message
	);
ELSE
	; // do nothing
END_CASE
END_METHOD

(*

## Short summary
This assertion method checks if the current string ``stringToCheck`` is length
is equal or grater than to ``minLength``

**Attention:** 
	All strings are handled as null terminated byte/word streams.
	For UTF-8 is end of the string 16#00
	For UTF-16 is end of the string 16#00_00

**Attention:** 
	The interface `IUnicodeAssertions` uses ``ANY_STRING``, 
	for this it's not possible to use literals/constants,
	because for ``ANY`` types generates the compiler ``__SYSTEM.AnyType``
	and ``__SYSTEM.AnyType`` contains a pointer  

.. <legal notes>

legal notes
=================
| SPDX-FileCopyrightText: © 2022 ekvip automation GmbH <info@ekvip.de>
| SPDX-License-Identifier: Apache-2.0
| For details check: Apache-2.0_

.. _Apache-2.0: https://www.apache.org/licenses/LICENSE-2.0

.. </legal notes>



*)

METHOD lengthIsMin
VAR_INPUT
	(* current string to check *)
	stringToCheck	:ANY_STRING;
	(* lower limit of the length of ``stringToCheck`` *)
	minLength		:UDINT;
	(* string length units of measurement *)
	stringLengthUnit	:UnicodeStringLengthUnit;
	(* message if the assertion is false *)
	message			:AssertMessage;
END_VAR
CASE stringToCheck.TypeClass OF
TYPE_CLASS.TYPE_STRING:
	THIS^.utf8Assertions.lengthIsMin(
		stringToCheck	:= stringToCheck.pValue,
		minLength		:= minLength,
		stringLengthUnit := stringLengthUnit,
		message			:= message
	);
TYPE_CLASS.TYPE_WSTRING:
	THIS^.utf16Assertions.lengthIsMin(
		stringToCheck	:= stringToCheck.pValue,
		minLength		:= minLength,
		stringLengthUnit := stringLengthUnit,
		message			:= message
	);
ELSE
	; // do nothing
END_CASE
END_METHOD

(*

## Short summary
This methods is the setter for the callback class if an assertion was false

.. <legal notes>

legal notes
=================
| SPDX-FileCopyrightText: © 2022 ekvip automation GmbH <info@ekvip.de>
| SPDX-License-Identifier: Apache-2.0
| For details check: Apache-2.0_

.. _Apache-2.0: https://www.apache.org/licenses/LICENSE-2.0

.. </legal notes>



*)

METHOD setCallBack
VAR_INPUT
	(* the class that must be informed if an assertion is false *)
	callBack	:IAssertCallBack;  
END_VAR
SUPER^.setCallBack(callBack);
THIS^.utf8Assertions.setCallBack(callBack);
THIS^.utf16Assertions.setCallBack(callBack);
END_METHOD

(*

## Short summary
This assertion method checks if the current string ``stringToCheck`` starts with ``start``

**Attention:** 
	All strings are handled as null terminated byte/word streams.
	For UTF-8 is end of the string 16#00
	For UTF-16 is end of the string 16#00_00

**Attention:** 
	The interface `IUnicodeAssertions` uses ``ANY_STRING``, 
	for this it's not possible to use literals/constants,
	because for ``ANY`` types generates the compiler ``__SYSTEM.AnyType``
	and ``__SYSTEM.AnyType`` contains a pointer  

**Attention:** 
	start of the string is **ALWAYS** the left side of the string 
	even for writings which written from right to left like Hebrew or Arabic

.. <legal notes>

legal notes
=================
| SPDX-FileCopyrightText: © 2022 ekvip automation GmbH <info@ekvip.de>
| SPDX-License-Identifier: Apache-2.0
| For details check: Apache-2.0_

.. _Apache-2.0: https://www.apache.org/licenses/LICENSE-2.0

.. </legal notes>



*)

METHOD startsWith
VAR_INPUT
	(* current string to check *)
	stringToCheck	:ANY_STRING;
	(* expected start of ``stringToCheck`` *)
	start			:ANY_STRING;
	(* message if the assertion is false *)
	message			:AssertMessage;
	(* ``TRUE`` means ignore cases; ``FALSE`` means cases must be equal too *)
	ignoreCases		:BOOL := FALSE;
	(* ``TRUE`` means truncation of spaces on the left side of ``stringToCheck``*)
	trim			:BOOL := FALSE;
	(*normalize both strings for check*)
	normalizeStrings :BOOL := TRUE;
END_VAR
IF ((
		stringToCheck.TypeClass <> start.TypeClass
	) OR_ELSE (
		stringToCheck.diSize = 0 
	) OR_ELSE ( 
		start.diSize = 0 
	)
) THEN
	THIS^.assertionWasWrong(message, THIS^.getDebugInfo('startsWith'));
	RETURN;
END_IF

CASE stringToCheck.TypeClass OF
TYPE_CLASS.TYPE_STRING:
	THIS^.utf8Assertions.startsWith(
		stringToCheck := stringToCheck.pValue,
		start := start.pValue,
		ignoreCases := ignoreCases,
		trim := trim,
		message := message,
		normalizeStrings := normalizeStrings
	);
TYPE_CLASS.TYPE_WSTRING:
	THIS^.utf16Assertions.startsWith(
		stringToCheck := stringToCheck.pValue,
		start := start.pValue,
		ignoreCases := ignoreCases,
		trim := trim,
		message := message,
		normalizeStrings := normalizeStrings
	);
ELSE
	; // do nothing
END_CASE
END_METHOD

END_FUNCTION_BLOCK

// ---- Assertor/Assertions/TimeAssertions/classes/TimeAssertions.TcPOU
(*

## Short summary
This class implements the interface `ITimeAssertions`.
It provides assertions for time data types
For ``LTIME`` assertions use `TimeAssertions.long`.
For ``TIME`` assertions use `TimeAssertions.simple`.


.. <legal notes>

legal notes
=================
| SPDX-FileCopyrightText: © 2022 ekvip automation GmbH <info@ekvip.de>
| SPDX-License-Identifier: Apache-2.0
| For details check: Apache-2.0_

.. _Apache-2.0: https://www.apache.org/licenses/LICENSE-2.0

.. </legal notes>

==

*)

{attribute 'reflection'}
FUNCTION_BLOCK INTERNAL TimeAssertions EXTENDS CNM_AbstractObject.Object IMPLEMENTS ITimeAssertions, IAssertCallBackSetter
VAR
	(* class to handle TIME assertions *)
	simpleTimeAssertions	:SimpleTimeAssertions();
	(* class to handle LTIME assertions *)
	longTimeAssertions		:LongTimeAssertions();
END_VAR

(*

## Short summary
This abstract property returns the class name of the concrete object, 
It's for debugging purpose

.. <legal notes>

legal notes
=================
| SPDX-FileCopyrightText: © 2022 ekvip automation GmbH <info@ekvip.de>
| SPDX-License-Identifier: Apache-2.0
| For details check: Apache-2.0_

.. _Apache-2.0: https://www.apache.org/licenses/LICENSE-2.0

.. </legal notes>

*)

PROPERTY className :CNM_AbstractObject.ClassName
GET
className := 'CNM_Assertor.TimeAssertions';
END_GET
END_PROPERTY

(*

## Short summary
Returns an interface (`I64BitTimeAssertions`)
with assert statements for 64 bit times 

.. <legal notes>

legal notes
=================
| SPDX-FileCopyrightText: © 2022 ekvip automation GmbH <info@ekvip.de>
| SPDX-License-Identifier: Apache-2.0
| For details check: Apache-2.0_

.. _Apache-2.0: https://www.apache.org/licenses/LICENSE-2.0

.. </legal notes>

*)

PROPERTY long :I64BitTimeAssertions
GET
long := THIS^.longTimeAssertions;
END_GET
END_PROPERTY

(*

## Short summary
This methods is the setter for the callback class if an assertion was false

.. <legal notes>

legal notes
=================
| SPDX-FileCopyrightText: © 2022 ekvip automation GmbH <info@ekvip.de>
| SPDX-License-Identifier: Apache-2.0
| For details check: Apache-2.0_

.. _Apache-2.0: https://www.apache.org/licenses/LICENSE-2.0

.. </legal notes>



*)

METHOD setCallBack
VAR_INPUT
	(* the class that must be informed if an assertion is false *)
	callBack	:IAssertCallBack;  
END_VAR
THIS^.simpleTimeAssertions.setCallBack(callBack);
THIS^.longTimeAssertions.setCallBack(callBack);
END_METHOD

(*

## Short summary
Returns an interface (`I32BitTimeAssertions`)
with assert statements for 32 bit times 

.. <legal notes>

legal notes
=================
| SPDX-FileCopyrightText: © 2022 ekvip automation GmbH <info@ekvip.de>
| SPDX-License-Identifier: Apache-2.0
| For details check: Apache-2.0_

.. _Apache-2.0: https://www.apache.org/licenses/LICENSE-2.0

.. </legal notes>

*)

PROPERTY simple :I32BitTimeAssertions
GET
simple := THIS^.simpleTimeAssertions;
END_GET
END_PROPERTY

END_FUNCTION_BLOCK

// ---- Assertor/Assertions/TimeAssertions/Time/classes/SimpleTimeAssertions.TcPOU
(*

## Short summary
This class implements the interface `I32BitTimeAssertions`. 
It contains the assert statements for the data type ``TIME``

.. <legal notes>

legal notes
=================
| SPDX-FileCopyrightText: © 2022 ekvip automation GmbH <info@ekvip.de>
| SPDX-License-Identifier: Apache-2.0
| For details check: Apache-2.0_

.. _Apache-2.0: https://www.apache.org/licenses/LICENSE-2.0

.. </legal notes>

==

*)

{attribute 'reflection'}
FUNCTION_BLOCK INTERNAL SimpleTimeAssertions EXTENDS AbstractAssertion IMPLEMENTS I32BitTimeAssertions
VAR CONSTANT
	(* maximum value for the data type ``TIME`` *)
	MAX_TIME	:TIME := TO_TIME(16#FF_FF_FF_FF);
END_VAR

(*

## Short summary
This abstract property returns the class name of the concrete object, 
It's for debugging purpose

.. <legal notes>

legal notes
=================
| SPDX-FileCopyrightText: © 2022 ekvip automation GmbH <info@ekvip.de>
| SPDX-License-Identifier: Apache-2.0
| For details check: Apache-2.0_

.. _Apache-2.0: https://www.apache.org/licenses/LICENSE-2.0

.. </legal notes>

*)

PROPERTY className :CNM_AbstractObject.ClassName
GET
className := 'CNM_Assertor.SimplyTimeAssertions';
END_GET
END_PROPERTY

(*

## Short summary
This method returns the passed time since the timestamp was created

.. <legal notes>

legal notes
=================
| SPDX-FileCopyrightText: © 2022 ekvip automation GmbH <info@ekvip.de>
| SPDX-License-Identifier: Apache-2.0
| For details check: Apache-2.0_

.. _Apache-2.0: https://www.apache.org/licenses/LICENSE-2.0

.. </legal notes>


:return: passed time since ``startTime``

*)

METHOD PROTECTED getTimePassed :TIME
VAR_INPUT
	(* timestamp start *)
	startTime	:TIME;
END_VAR
VAR
	(* current time to calculate the passed time *)
	currentTime	:TIME;
END_VAR
currentTime := TIME();
IF (currentTime > startTime) THEN
	getTimePassed := (currentTime - startTime);
ELSE
	getTimePassed := ((THIS^.MAX_TIME - startTime) + currentTime);
END_IF
END_METHOD

(*

## Short summary
This assertion method checks whether time has elapsed since the timestamp time

.. <legal notes>

legal notes
=================
| SPDX-FileCopyrightText: © 2022 ekvip automation GmbH <info@ekvip.de>
| SPDX-License-Identifier: Apache-2.0
| For details check: Apache-2.0_

.. _Apache-2.0: https://www.apache.org/licenses/LICENSE-2.0

.. </legal notes>



*)

METHOD timeHasExpired
VAR_INPUT
	(* start time you get it with ``TIME()`` *)
	timestamp		:TIME;
	(* timeout like ``t#300ms`` *)
	expiringTime	:TIME;
	(* message if the assertion is false *)
	message			:AssertMessage;
END_VAR
VAR
	(* measured passed time *)
	passedTime		:TIME;
END_VAR
passedTime := THIS^.getTimePassed(timestamp);
IF (passedTime < expiringTime) THEN
	THIS^.assertionWasWrong(
		message			:= message,
		additionalText	:= THIS^.getDebugInfo('timeHasExpired')
	);	
END_IF
END_METHOD

(*

## Short summary
This assertion method checks that the time since the timestamp time has not yet elapsed

.. <legal notes>

legal notes
=================
| SPDX-FileCopyrightText: © 2022 ekvip automation GmbH <info@ekvip.de>
| SPDX-License-Identifier: Apache-2.0
| For details check: Apache-2.0_

.. _Apache-2.0: https://www.apache.org/licenses/LICENSE-2.0

.. </legal notes>



*)

METHOD timeHasNotExpired
VAR_INPUT
	(* start time you get it with ``TIME()`` *)
	timestamp		:TIME;
	(* timeout like ``t#300ms`` *)
	expiringTime	:TIME;
	(* message if the assertion is false *)
	message			:AssertMessage;
END_VAR
VAR
	(* measured passed time *)
	passedTime		:TIME;
END_VAR
passedTime := THIS^.getTimePassed(timestamp);
IF (passedTime >= expiringTime) THEN
	THIS^.assertionWasWrong(
		message			:= message,
		additionalText	:= THIS^.getDebugInfo('timeHasNotExpired')
	);	
END_IF
END_METHOD

(*

## Short summary
This assertion method checks if the current value is equal to the expected value

.. <legal notes>

legal notes
=================
| SPDX-FileCopyrightText: © 2022 ekvip automation GmbH <info@ekvip.de>
| SPDX-License-Identifier: Apache-2.0
| For details check: Apache-2.0_

.. _Apache-2.0: https://www.apache.org/licenses/LICENSE-2.0

.. </legal notes>



*)

METHOD valueIsEqualTo
VAR_INPUT
	(* current value to check *)
	currentValue	:TIME;
	(* expected value to compare *)
	expectedValue	:TIME;
	(* message if the assertion is false *)
	message			:AssertMessage;
END_VAR
IF (currentValue <> expectedValue) THEN
	THIS^.assertionWasWrong(
		message			:= message,
		additionalText	:= THIS^.getDebugInfo('valueIsEqualTo')
	);	
END_IF
END_METHOD

(*

## Short summary
This assertion method checks if the current value is greater than the less value

.. <legal notes>

legal notes
=================
| SPDX-FileCopyrightText: © 2022 ekvip automation GmbH <info@ekvip.de>
| SPDX-License-Identifier: Apache-2.0
| For details check: Apache-2.0_

.. _Apache-2.0: https://www.apache.org/licenses/LICENSE-2.0

.. </legal notes>



*)

METHOD valueIsGreaterThan
VAR_INPUT
	(* current value to check *)
	currentValue	:TIME;
	(* less than lower limit *)
	lessValue		:TIME;
	(* message if the assertion is false *)
	message			:AssertMessage;
END_VAR
IF (currentValue <= lessValue) THEN
	THIS^.assertionWasWrong(
		message			:= message,
		additionalText	:= THIS^.getDebugInfo('valueIsGreaterThan')
	);	
END_IF
END_METHOD

(*

## Short summary
This assertion method checks if the current value is inside a limit

**Attention:** 
	limits are included: ``valueIsInRangeOf(t#3ms,t#3ms ,t#3ms)`` is a true assertion

.. <legal notes>

legal notes
=================
| SPDX-FileCopyrightText: © 2022 ekvip automation GmbH <info@ekvip.de>
| SPDX-License-Identifier: Apache-2.0
| For details check: Apache-2.0_

.. _Apache-2.0: https://www.apache.org/licenses/LICENSE-2.0

.. </legal notes>



*)

METHOD valueIsInRangeOf
VAR_INPUT
	(* lower limit for the current value *)
	lowerLimit		:TIME;
	(* current value to check *)
	currentValue	:TIME;
	(* upper limit for the current value *)
	upperLimit		:TIME;
	(* message if the assertion is false *)
	message			:AssertMessage;
END_VAR
IF ((currentValue < lowerLimit) OR (currentValue > upperLimit)) THEN
	THIS^.assertionWasWrong(
		message			:= message,
		additionalText	:= THIS^.getDebugInfo('valueIsInRangeOf')
	);	
END_IF
END_METHOD

(*

## Short summary
This assertion method checks if the current value is less than the greater value

.. <legal notes>

legal notes
=================
| SPDX-FileCopyrightText: © 2022 ekvip automation GmbH <info@ekvip.de>
| SPDX-License-Identifier: Apache-2.0
| For details check: Apache-2.0_

.. _Apache-2.0: https://www.apache.org/licenses/LICENSE-2.0

.. </legal notes>



*)

METHOD valueIsLessThan
VAR_INPUT
	(* current value to check *)
	currentValue	:TIME;
	(* greater than upper limit *)
	greaterValue	:TIME;
	(* message if the assertion is false *)
	message			:AssertMessage;
END_VAR
IF (currentValue >= greaterValue) THEN
	THIS^.assertionWasWrong(
		message			:= message,
		additionalText	:= THIS^.getDebugInfo('valueIsLessThan')
	);	
END_IF
END_METHOD

(*

## Short summary
This assertion method checks if the current value is less than or equal to the maximum value

.. <legal notes>

legal notes
=================
| SPDX-FileCopyrightText: © 2022 ekvip automation GmbH <info@ekvip.de>
| SPDX-License-Identifier: Apache-2.0
| For details check: Apache-2.0_

.. _Apache-2.0: https://www.apache.org/licenses/LICENSE-2.0

.. </legal notes>



*)

METHOD valueIsMax
VAR_INPUT
	(* current value to check *)
	currentValue	:TIME;
	(* upper limit for the current value *)
	maximumValue	:TIME;
	(* message if the assertion is false *)
	message			:AssertMessage;
END_VAR
IF (currentValue > maximumValue) THEN
	THIS^.assertionWasWrong(
		message			:= message,
		additionalText	:= THIS^.getDebugInfo('valueIsMax')
	);	
END_IF
END_METHOD

(*

## Short summary
This assertion method checks if the current value is greater than or equal to the minimum value

.. <legal notes>

legal notes
=================
| SPDX-FileCopyrightText: © 2022 ekvip automation GmbH <info@ekvip.de>
| SPDX-License-Identifier: Apache-2.0
| For details check: Apache-2.0_

.. _Apache-2.0: https://www.apache.org/licenses/LICENSE-2.0

.. </legal notes>



*)

METHOD valueIsMin
VAR_INPUT
	(* current value to check *)
	currentValue	:TIME;
	(* lower limit for the current value *)
	minimumValue	:TIME;
	(* message if the assertion is false *)
	message			:AssertMessage;
END_VAR
IF (currentValue < minimumValue) THEN
	THIS^.assertionWasWrong(
		message			:= message,
		additionalText	:= THIS^.getDebugInfo('valueIsMin')
	);	
END_IF
END_METHOD

(*

## Short summary
This assertion method checks if the current value is not equal to the unexpected value

.. <legal notes>

legal notes
=================
| SPDX-FileCopyrightText: © 2022 ekvip automation GmbH <info@ekvip.de>
| SPDX-License-Identifier: Apache-2.0
| For details check: Apache-2.0_

.. _Apache-2.0: https://www.apache.org/licenses/LICENSE-2.0

.. </legal notes>



*)

METHOD valueIsNotEqualTo
VAR_INPUT
	(* current value to check *)
	currentValue	:TIME;
	(* unexpected value to compare *)
	unexpectedValue	:TIME;
	(* message if the assertion is false *)
	message			:AssertMessage;
END_VAR
IF (currentValue = unexpectedValue) THEN
	THIS^.assertionWasWrong(
		message			:= message,
		additionalText	:= THIS^.getDebugInfo('valueIsNotEqualTo')
	);	
END_IF
END_METHOD

END_FUNCTION_BLOCK

// ---- Assertor/Assertions/TimeAssertions/LTime/classes/LongTimeAssertions.TcPOU
(*

## Short summary
This class implements the interface `I64BitTimeAssertions`. 
It provides the assert statements for the data type ``LTIME``

.. <legal notes>

legal notes
=================
| SPDX-FileCopyrightText: © 2022 ekvip automation GmbH <info@ekvip.de>
| SPDX-License-Identifier: Apache-2.0
| For details check: Apache-2.0_

.. _Apache-2.0: https://www.apache.org/licenses/LICENSE-2.0

.. </legal notes>

==

*)

{attribute 'reflection'}
FUNCTION_BLOCK INTERNAL LongTimeAssertions EXTENDS AbstractAssertion IMPLEMENTS I64BitTimeAssertions
VAR CONSTANT
	(* maximum value for the data type ``LTIME`` *)
	MAX_TIME	:LTIME := TO_LTIME(16#FFFF_FFFF_FFFF_FFFF);
END_VAR

(*

## Short summary
This abstract property returns the class name of the concrete object, 
It's for debugging purpose

.. <legal notes>

legal notes
=================
| SPDX-FileCopyrightText: © 2022 ekvip automation GmbH <info@ekvip.de>
| SPDX-License-Identifier: Apache-2.0
| For details check: Apache-2.0_

.. _Apache-2.0: https://www.apache.org/licenses/LICENSE-2.0

.. </legal notes>

*)

PROPERTY className :CNM_AbstractObject.ClassName
GET
className := 'CNM_Assertor.LongTimeAssertions';
END_GET
END_PROPERTY

(*

## Short summary
This method returns the passed time since the timestamp was created

.. <legal notes>

legal notes
=================
| SPDX-FileCopyrightText: © 2022 ekvip automation GmbH <info@ekvip.de>
| SPDX-License-Identifier: Apache-2.0
| For details check: Apache-2.0_

.. _Apache-2.0: https://www.apache.org/licenses/LICENSE-2.0

.. </legal notes>


:return: passed time since ``startTime``

*)

METHOD PROTECTED getTimePassed :LTIME
VAR_INPUT
	(* timestamp start *)
	startTime	:LTIME;
END_VAR
VAR
	(* current time to calculate the passed time *)
	currentTime	:LTIME;
END_VAR
currentTime := LTIME();
IF (currentTime > startTime) THEN
	getTimePassed := (currentTime - startTime);
ELSE
	getTimePassed := ((THIS^.MAX_TIME - startTime) + currentTime);
END_IF
END_METHOD

(*

## Short summary
This assertion method checks whether time has elapsed since the timestamp time

.. <legal notes>

legal notes
=================
| SPDX-FileCopyrightText: © 2022 ekvip automation GmbH <info@ekvip.de>
| SPDX-License-Identifier: Apache-2.0
| For details check: Apache-2.0_

.. _Apache-2.0: https://www.apache.org/licenses/LICENSE-2.0

.. </legal notes>



*)

METHOD timeHasExpired
VAR_INPUT
	(* start time you get it with ``LTIME()`` *)
	timestamp		:LTIME;
	(* timeout like ``lt#300ms`` *)
	expiringTime	:LTIME;
	(* message if the assertion is false *)
	message			:AssertMessage;
END_VAR
VAR
	(* measured passed time *)
	passedTime		:LTIME;
END_VAR
passedTime := THIS^.getTimePassed(timestamp);
IF (passedTime < expiringTime) THEN
	THIS^.assertionWasWrong(
		message			:= message,
		additionalText	:= THIS^.getDebugInfo('timeHasExpired')
	);	
END_IF
END_METHOD

(*

## Short summary
This assertion method checks that the time since the timestamp time has not yet elapsed

.. <legal notes>

legal notes
=================
| SPDX-FileCopyrightText: © 2022 ekvip automation GmbH <info@ekvip.de>
| SPDX-License-Identifier: Apache-2.0
| For details check: Apache-2.0_

.. _Apache-2.0: https://www.apache.org/licenses/LICENSE-2.0

.. </legal notes>



*)

METHOD timeHasNotExpired
VAR_INPUT
	(* start time you get it with ``LTIME()`` *)
	timestamp		:LTIME;
	(* timeout like ``lt#300ms`` *)
	expiringTime	:LTIME;
	(* message if the assertion is false *)
	message			:AssertMessage;
END_VAR
VAR
	(* measured passed time *)
	passedTime		:LTIME;
END_VAR
passedTime := THIS^.getTimePassed(timestamp);
IF (passedTime >= expiringTime) THEN
	THIS^.assertionWasWrong(
		message			:= message,
		additionalText	:= THIS^.getDebugInfo('timeHasNotExpired')
	);	
END_IF
END_METHOD

(*

## Short summary
This assertion method checks if the current value is equal to the expected value

.. <legal notes>

legal notes
=================
| SPDX-FileCopyrightText: © 2022 ekvip automation GmbH <info@ekvip.de>
| SPDX-License-Identifier: Apache-2.0
| For details check: Apache-2.0_

.. _Apache-2.0: https://www.apache.org/licenses/LICENSE-2.0

.. </legal notes>



*)

METHOD valueIsEqualTo
VAR_INPUT
	(* current value to check *)
	currentValue	:LTIME;
	(* expected value to compare *)
	expectedValue	:LTIME;
	(* message if the assertion is false *)
	message	:AssertMessage;
END_VAR
IF (currentValue <> expectedValue) THEN
	THIS^.assertionWasWrong(
		message			:= message,
		additionalText	:= THIS^.getDebugInfo('valueIsEqualTo')
	);	
END_IF
END_METHOD

(*

## Short summary
This assertion method checks if the current value is greater than the less value

.. <legal notes>

legal notes
=================
| SPDX-FileCopyrightText: © 2022 ekvip automation GmbH <info@ekvip.de>
| SPDX-License-Identifier: Apache-2.0
| For details check: Apache-2.0_

.. _Apache-2.0: https://www.apache.org/licenses/LICENSE-2.0

.. </legal notes>



*)

METHOD valueIsGreaterThan
VAR_INPUT
	(* current value to check *)
	currentValue	:LTIME;
	(* less than lower limit *)
	lessValue		:LTIME;
	(* message if the assertion is false *)
	message	: AssertMessage;
END_VAR
IF (currentValue <= lessValue) THEN
	THIS^.assertionWasWrong(
		message			:= message,
		additionalText	:= THIS^.getDebugInfo('valueIsGreaterThan')
	);	
END_IF
END_METHOD

(*

## Short summary
This assertion method checks if the current value is inside a limit

**Attention:** 
	limits are included: ``valueIsInRangeOf(t#3ms,t#3ms ,t#3ms)`` is a true assertion

.. <legal notes>

legal notes
=================
| SPDX-FileCopyrightText: © 2022 ekvip automation GmbH <info@ekvip.de>
| SPDX-License-Identifier: Apache-2.0
| For details check: Apache-2.0_

.. _Apache-2.0: https://www.apache.org/licenses/LICENSE-2.0

.. </legal notes>



*)

METHOD valueIsInRangeOf
VAR_INPUT
	(* lower limit for the current value *)
	lowerLimit		:LTIME;
	(* current value to check *)
	currentValue	:LTIME;
	(* upper limit for the current value *)
	upperLimit		:LTIME;
	(* message if the assertion is false *)
	message			:AssertMessage;
END_VAR
VAR
	(* additional information for the callback function *)
	additionalText	:Tc2_System.T_MaxString;
END_VAR
IF ((currentValue < lowerLimit) OR (currentValue > upperLimit)) THEN
	THIS^.assertionWasWrong(
		message			:= message,
		additionalText	:= THIS^.getDebugInfo('valueIsInRangeOf')
	);	
END_IF
END_METHOD

(*

## Short summary
This assertion method checks if the current value is less than the greater value

.. <legal notes>

legal notes
=================
| SPDX-FileCopyrightText: © 2022 ekvip automation GmbH <info@ekvip.de>
| SPDX-License-Identifier: Apache-2.0
| For details check: Apache-2.0_

.. _Apache-2.0: https://www.apache.org/licenses/LICENSE-2.0

.. </legal notes>



*)

METHOD valueIsLessThan
VAR_INPUT
	(* current value to check *)
	currentValue	:LTIME;
	(* greater than upper limit *)
	greaterValue	:LTIME;
	(* message if the assertion is false *)
	message			:AssertMessage;
END_VAR
IF (currentValue >= greaterValue) THEN
	THIS^.assertionWasWrong(
		message			:= message,
		additionalText	:= THIS^.getDebugInfo('valueIsLessThan')
	);	
END_IF
END_METHOD

(*

## Short summary
This assertion method checks if the current value is less than or equal to the maximum value

.. <legal notes>

legal notes
=================
| SPDX-FileCopyrightText: © 2022 ekvip automation GmbH <info@ekvip.de>
| SPDX-License-Identifier: Apache-2.0
| For details check: Apache-2.0_

.. _Apache-2.0: https://www.apache.org/licenses/LICENSE-2.0

.. </legal notes>



*)

METHOD valueIsMax
VAR_INPUT
	(* current value to check *)
	currentValue	:LTIME;
	(* upper limit for the current value *)
	maximumValue	:LTIME;
	(* message if the assertion is false *)
	message			:AssertMessage;
END_VAR
IF (currentValue > maximumValue) THEN
	THIS^.assertionWasWrong(
		message			:= message,
		additionalText	:= THIS^.getDebugInfo('valueIsMax')
	);	
END_IF
END_METHOD

(*

## Short summary
This assertion method checks if the current value is greater than or equal to the minimum value

.. <legal notes>

legal notes
=================
| SPDX-FileCopyrightText: © 2022 ekvip automation GmbH <info@ekvip.de>
| SPDX-License-Identifier: Apache-2.0
| For details check: Apache-2.0_

.. _Apache-2.0: https://www.apache.org/licenses/LICENSE-2.0

.. </legal notes>



*)

METHOD valueIsMin
VAR_INPUT
	(* current value to check *)
	currentValue	:LTIME;
	(* lower limit for the current value *)
	minimumValue	:LTIME;
	(* message if the assertion is false *)
	message			:AssertMessage;
END_VAR
IF (currentValue < minimumValue) THEN
	THIS^.assertionWasWrong(
		message			:= message,
		additionalText	:= THIS^.getDebugInfo('valueIsMin')
	);	
END_IF
END_METHOD

(*

## Short summary
This assertion method checks if the current value is not equal to the unexpected value

.. <legal notes>

legal notes
=================
| SPDX-FileCopyrightText: © 2022 ekvip automation GmbH <info@ekvip.de>
| SPDX-License-Identifier: Apache-2.0
| For details check: Apache-2.0_

.. _Apache-2.0: https://www.apache.org/licenses/LICENSE-2.0

.. </legal notes>



*)

METHOD valueIsNotEqualTo
VAR_INPUT
	(* current value to check *)
	currentValue	:LTIME;
	(* unexpected value to compare *)
	unexpectedValue	:LTIME;
	(* message if the assertion is false *)
	message			:AssertMessage;
END_VAR
IF (currentValue = unexpectedValue) THEN
	THIS^.assertionWasWrong(
		message			:= message,
		additionalText	:= THIS^.getDebugInfo('valueIsNotEqualTo')
	);	
END_IF
END_METHOD

END_FUNCTION_BLOCK

// ---- Assertor/classes/AbstractAssertor.TcPOU
(*

## Short summary

This abstract class provides assert statements in a `fluent interface`_ style for the most common data types. 
It implements the interfaces `IAssertor` and `IAssertCallBack`
If you need assertion statements you've to extend this class and you've to overwrite the methods
`AbstractAssertor.assertionWasWrong`
`AbstractAssertor.className`

.. _`fluent interface`: https://en.wikipedia.org/wiki/Fluent_interface

.. <legal notes>

legal notes
=================
| SPDX-FileCopyrightText: © 2022 ekvip automation GmbH <info@ekvip.de>
| SPDX-License-Identifier: Apache-2.0
| For details check: Apache-2.0_

.. _Apache-2.0: https://www.apache.org/licenses/LICENSE-2.0

.. </legal notes>



*)

{attribute 'reflection'}
FUNCTION_BLOCK ABSTRACT AbstractAssertor EXTENDS CNM_AbstractObject.Object IMPLEMENTS IAssertor, IAssertCallBack
VAR
	(* class to handle all the worth assertions *)
	{attribute 'hide'}
	assertions	:Assertions();
END_VAR

(*

## Short summary
Returns the interface `IAssertions`
to get access to the assert statements

.. <legal notes>

legal notes
=================
| SPDX-FileCopyrightText: © 2022 ekvip automation GmbH <info@ekvip.de>
| SPDX-License-Identifier: Apache-2.0
| For details check: Apache-2.0_

.. _Apache-2.0: https://www.apache.org/licenses/LICENSE-2.0

.. </legal notes>



*)

PROPERTY assert :IAssertions
GET
assert := THIS^.assertions;
END_GET
END_PROPERTY

(*

## Short summary
This method is called if an assertion was ``FALSE``

.. <legal notes>

legal notes
=================
| SPDX-FileCopyrightText: © 2022 ekvip automation GmbH <info@ekvip.de>
| SPDX-License-Identifier: Apache-2.0
| For details check: Apache-2.0_

.. _Apache-2.0: https://www.apache.org/licenses/LICENSE-2.0

.. </legal notes>



*)

METHOD ABSTRACT assertionWasWrong
VAR_INPUT
	(* caller object of the method *)
	caller			:CNM_AbstractObject.IObject;
	(* alarm message *)
	message			:AssertMessage;
	(* debugging information *) 
	additionalText	:Tc2_System.T_MaxString;
END_VAR
END_METHOD

(*

## Short summary
This abstract property returns the class name of the concrete object, 
It's for debugging purpose

**Attention:** 
	For derivations: **It is necessary that this property is overridden by the concrete class**

.. <legal notes>

legal notes
=================
| SPDX-FileCopyrightText: © 2022 ekvip automation GmbH <info@ekvip.de>
| SPDX-License-Identifier: Apache-2.0
| For details check: Apache-2.0_

.. _Apache-2.0: https://www.apache.org/licenses/LICENSE-2.0

.. </legal notes>

*)

PROPERTY ABSTRACT className :CNM_AbstractObject.ClassName
GET
END_GET
END_PROPERTY

(*

## Short summary
The constructor ``FB_init`` is needed to create an unique hash code.
The hash code is a pseudo random number create with a [xorshift](https://en.wikipedia.org/wiki/Xorshift) algorithm.
It can be overwritten on derivations, because it will be called implicit, ``SUPER^.FB_init()`` is not required.
For more information check: [Behavoir with derived function blocks](https://infosys.beckhoff.com/content/1033/tc3_plc_intro/5482088715.html?id=6983869892358031022)

.. <legal notes>

legal notes
=================
| SPDX-FileCopyrightText: © 2022 ekvip automation GmbH <info@ekvip.de>
| SPDX-License-Identifier: Apache-2.0
| For details check: Apache-2.0_

.. _Apache-2.0: https://www.apache.org/licenses/LICENSE-2.0

.. </legal notes>



*)

METHOD FB_init :BOOL;
VAR_INPUT
	(* if TRUE, the retain variables are initialized (warm start / cold start)*)
	bInitRetains	:BOOL;
	(* if TRUE, the instance afterwards gets moved into the copy code (online change) *)
	bInCopyCode		:BOOL;  
END_VAR
VAR
	{attribute 'hide'}
	newHashstate3		:CNM_AbstractObject.Hashcode;
END_VAR
VAR CONSTANT
	{attribute 'hide'}
	NUMBER_OF_LEFT_SHIFTS		:UINT	:= 17;
	{attribute 'hide'}
	NUMBER_OF_LEFT_ROTATIONS	:UINT   := 45;
END_VAR
THIS^.assertions.setCallBack(THIS^);
END_METHOD

END_FUNCTION_BLOCK

// ---- Project Information/F_GetCompany.TcPOU
// This function has been automatically generated from the project information.
{attribute 'signature_flag' := '1073741824'}
{attribute 'TcGenerated'}
{attribute 'no-analysis'}
FUNCTION F_GetCompany : WSTRING
VAR_INPUT
	
END_VAR

F_GetCompany := "ekvip automation GmbH";

END_FUNCTION

// ---- Project Information/F_GetTitle.TcPOU
// This function has been automatically generated from the project information.
{attribute 'signature_flag' := '1073741824'}
{attribute 'TcGenerated'}
{attribute 'no-analysis'}
FUNCTION F_GetTitle : WSTRING
VAR_INPUT
	
END_VAR

F_GetTitle := "CNM_AssertionInterfaces";

END_FUNCTION

// ---- Project Information/F_GetVersion.TcPOU
// This function has been automatically generated from the project information.
{attribute 'signature_flag' := '1073741824'}
{attribute 'TcGenerated'}
{attribute 'no-analysis'}
FUNCTION F_GetVersion : ST_LibVersion
VAR_INPUT
	
END_VAR

F_GetVersion.iMajor := 0;
F_GetVersion.iMinor := 1;
F_GetVersion.iBuild := 1;
F_GetVersion.iRevision := 0;
F_GetVersion.sVersion := '0.1.1.0';
F_GetVersion.nFlags := 0;

END_FUNCTION
